FUNCTION_BLOCK FB_SubNestedView EXTENDS FB_BA_View
VAR_INPUT CONSTANT
	SubView		: FB_NestedView		:= (View := (iParent:=THIS^));
END_VAR

SUPER^();

SubView();

END_FUNCTION_BLOCK

(* stored: Version 1.1.0.1, ProductVersion 3.1.4024.5
   POU FB_SubNestedView: Id {28a2423f-9859-4454-ab25-9c96d035c721}, SpecialFunc None *)
